# EPICS substitutions: vacuum/MAIN_TRUNK/db/l426_agilent4uhv.substitutions
# Agilent4UHV substitutions file

file db/agilent4uhv.db
{
     pattern {LOCA,			DEV,			PORT,		ADDR,	TIMEOUT}
     		{HL4,			VL426_1,		4uhv_1,		0,		0.2}
     		{HL4,			VL426_2,		4uhv_2,		0,		0.2}
}

file db/agilent4uhv_alias.db
{
     pattern {LOCA,			DEV,			SUB1,				SUB2,				SUB3,					SUB4,				PORT,		ADDR,	TIMEOUT}
     		 {HL4,			VL426_1,		IP01:L426_Acc601,		IP02:L426_Acc602,		IP03:L426_Acc603,			IP04:L426_Acc604,		4uhv_1,		0,		0.2}
		 {HL4,			VL426_2,		IP05:L426_Acc605,		IP06:L426_Wave601,	IP07:L426_Kly601,			IP08:Empty,			4uhv_2,		0,		0.2}
}
